{attribute 'qualified_only'}
{attribute 'strict'}
{attribute 'to_string'}
TYPE E_DrukknoppenStatus :
(
	StartKnop := 0,
	StopKnop,
	ResetKnop
);
END_TYPE

(* stored: Version 1.1.0.1
   DUT E_DrukknoppenStatus: Id {752a2515-1a0f-458a-8578-c36c76913157} *)
